SUBAPPLICATION HW_1Sensor (* Subapplication Type *)
  (* Standard: 61499-2 *)
  (* Version 1.0, 2020-07-20, dummy *)
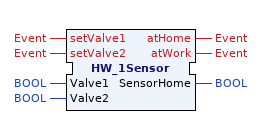
  EVENT_INPUT
    setValve1;
    setValve2;
  END_EVENT
  EVENT_OUTPUT
    atHome;
    atWork;
  END_EVENT
  VAR_INPUT
    Valve1 : BOOL;
    Valve2 : BOOL;
  END_VAR
  VAR_OUTPUT
    SensorHome : BOOL;
  END_VAR
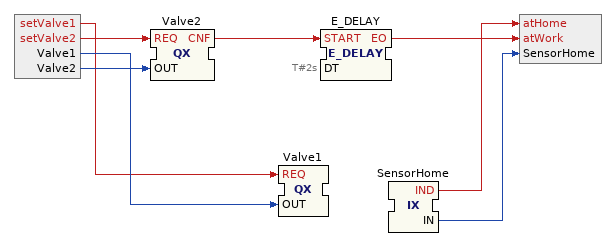
  FBS
    Valve1 : QX;
    SensorHome : IX;
    Valve2 : QX;
    E_DELAY : E_DELAY(DT := T#2s);
  END_FBS
  EVENT_CONNECTIONS
    setValve1 TO Valve1.REQ;
    setValve2 TO Valve2.REQ;
    Valve2.CNF TO E_DELAY.START;
    E_DELAY.EO TO atWork;
    SensorHome.IND TO atHome;
  END_CONNECTIONS
  DATA_CONNECTIONS
    Valve1 TO Valve1.OUT;
    Valve2 TO Valve2.OUT;
    SensorHome.IN TO SensorHome;
  END_CONNECTIONS
END_SUBAPPLICATION
